        //********************************************
        // Device name: TS2-010CRM:WtrC-YCV-103
        // Device type: ICS_PV
        //********************************************

      "DEV_TS2-010CRM:WtrC-YCV-103_iDB" (EPICSToPLCLength:=5,
      EPICSToPLCDataBlockOffset:=55,
      PLCToEPICSLength:=34,
      PLCToEPICSDataBlockOffset:=137);

        //********************************************
        // Device name: TS2-010CRM:WtrC-YCV-104
        // Device type: ICS_PV
        //********************************************

      "DEV_TS2-010CRM:WtrC-YCV-104_iDB" (EPICSToPLCLength:=5,
      EPICSToPLCDataBlockOffset:=60,
      PLCToEPICSLength:=34,
      PLCToEPICSDataBlockOffset:=171);

        //********************************************
        // Device name: TS2-010CRM:WtrC-YSV-109
        // Device type: ICS_PV
        //********************************************

      "DEV_TS2-010CRM:WtrC-YSV-109_iDB" (EPICSToPLCLength:=5,
      EPICSToPLCDataBlockOffset:=65,
      PLCToEPICSLength:=34,
      PLCToEPICSDataBlockOffset:=205);

        //********************************************
        // Device name: TS2-010CRM:WtrC-YSV-110
        // Device type: ICS_PV
        //********************************************

      "DEV_TS2-010CRM:WtrC-YSV-110_iDB" (EPICSToPLCLength:=5,
      EPICSToPLCDataBlockOffset:=70,
      PLCToEPICSLength:=34,
      PLCToEPICSDataBlockOffset:=239);

        //********************************************
        // Device name: TS2-010CRM:WtrC-YSV-111
        // Device type: ICS_PV
        //********************************************

      "DEV_TS2-010CRM:WtrC-YSV-111_iDB" (EPICSToPLCLength:=5,
      EPICSToPLCDataBlockOffset:=75,
      PLCToEPICSLength:=34,
      PLCToEPICSDataBlockOffset:=273);

        //********************************************
        // Device name: TS2-010CRM:WtrC-YSV-112
        // Device type: ICS_PV
        //********************************************

      "DEV_TS2-010CRM:WtrC-YSV-112_iDB" (EPICSToPLCLength:=5,
      EPICSToPLCDataBlockOffset:=80,
      PLCToEPICSLength:=34,
      PLCToEPICSDataBlockOffset:=307);

        //********************************************
        // Device name: TS2-010CRM:WtrC-YSV-113
        // Device type: ICS_PV
        //********************************************

      "DEV_TS2-010CRM:WtrC-YSV-113_iDB" (EPICSToPLCLength:=5,
      EPICSToPLCDataBlockOffset:=85,
      PLCToEPICSLength:=34,
      PLCToEPICSDataBlockOffset:=341);

        //********************************************
        // Device name: TS2-010CRM:WtrC-TE-101
        // Device type: ICS_TT
        //********************************************

      "DEV_TS2-010CRM:WtrC-TE-101_iDB" (EPICSToPLCLength:=15,
      EPICSToPLCDataBlockOffset:=90,
      PLCToEPICSLength:=29,
      PLCToEPICSDataBlockOffset:=375);

        //********************************************
        // Device name: TS2-010CRM:WtrC-TE-102
        // Device type: ICS_TT
        //********************************************

      "DEV_TS2-010CRM:WtrC-TE-102_iDB" (EPICSToPLCLength:=15,
      EPICSToPLCDataBlockOffset:=105,
      PLCToEPICSLength:=29,
      PLCToEPICSDataBlockOffset:=404);

        //********************************************
        // Device name: TS2-010CRM:WtrC-TE-103
        // Device type: ICS_TT
        //********************************************

      "DEV_TS2-010CRM:WtrC-TE-103_iDB" (EPICSToPLCLength:=15,
      EPICSToPLCDataBlockOffset:=120,
      PLCToEPICSLength:=29,
      PLCToEPICSDataBlockOffset:=433);

        //********************************************
        // Device name: TS2-010CRM:WtrC-TE-104
        // Device type: ICS_TT
        //********************************************

      "DEV_TS2-010CRM:WtrC-TE-104_iDB" (EPICSToPLCLength:=15,
      EPICSToPLCDataBlockOffset:=135,
      PLCToEPICSLength:=29,
      PLCToEPICSDataBlockOffset:=462);
END_FUNCTION
DATA_BLOCK "EPICS_DebuggerResult"
{ S7_Optimized_Access := 'TRUE' }
VERSION : 0.1
NON_RETAIN
   VAR
      EPICS_Debugger_UtilitiesCall : String;   // PLCFactory Utilities call status
      EPICS_Debugger_DeviceCalls : String;   // PLCFactory DeviceCalls status
      EPICS_Debugger_IOCHash : String;   // EPICS IOC Hash vs. PLCFactory Hash
      EPICS_Debugger_ModBusHeartBeat : String;   // EPICS IOC Modbus (IOC->PLC) communication status
      EPICS_Debugger_S7Connection : String;   // EPICS IOC S7 TCP (PLC->IOC) communication status
      EPICS_Debugger_EPICS_GeneralState : String;   // Main status of the EPICS IOC communication
      EPICS_S7Port : Int;   // Actual TCP port that has been opened by the PLC
      EPICS_ModbusPort : Int;   // Actual ModBusTCP port that has been opened by the PLC
      EPICS_PLC_EthernetInterface : UInt;   // The currently used HW Identifer of the Ethernet Port on the PLC dedicated to EPICS
      EPICS_PayloadSize_InBytes : UInt;   // The currently configured payload size in bytes
      EPICS_PLC_Hash : DInt;   // The PLC Hash
      EPICS_PLCFactory_Version : String;   // The PLCFactory version that was used to generate the PLC code
      EPICS_CommunicationOK : Bool;   // Overall EPICS communication is OK
   END_VAR

BEGIN

END_DATA_BLOCK
FUNCTION_BLOCK "EPICS_DebuggerFB"
{ S7_Optimized_Access := 'TRUE' }
VERSION : 0.1
   VAR
      CheckUtilitiesTON {OriginalPartName := 'IEC_TIMER'; LibVersion := '1.0'; ExternalAccessible := 'False'; ExternalVisible := 'False'; ExternalWritable := 'False'} : TON_TIME;
      UtilSquareErrorTON { ExternalAccessible := 'False'; ExternalVisible := 'False'; ExternalWritable := 'False'} : Bool;
      CheckUtilitiesTON2 {OriginalPartName := 'IEC_TIMER'; LibVersion := '1.0'; ExternalAccessible := 'False'; ExternalVisible := 'False'; ExternalWritable := 'False'} : TON_TIME;
      UtilSquareErrorTON2 { ExternalAccessible := 'False'; ExternalVisible := 'False'; ExternalWritable := 'False'} : Bool;
      ModBus_TON {OriginalPartName := 'IEC_TIMER'; LibVersion := '1.0'; ExternalAccessible := 'False'; ExternalVisible := 'False'; ExternalWritable := 'False'} : TON_TIME;
      ModBus_wordsave { ExternalAccessible := 'False'; ExternalVisible := 'False'; ExternalWritable := 'False'} : Word;
   END_VAR
   VAR DB_SPECIFIC
      Helper_String { ExternalAccessible := 'False'; ExternalVisible := 'False'; ExternalWritable := 'False'} : String;
      Helper_String_Array { ExternalAccessible := 'False'; ExternalVisible := 'False'; ExternalWritable := 'False'} AT Helper_String : Struct
         String_Maximal { ExternalAccessible := 'False'; ExternalVisible := 'False'; ExternalWritable := 'False'} : Byte;
         String_Actual { ExternalAccessible := 'False'; ExternalVisible := 'False'; ExternalWritable := 'False'} : Byte;
         StringValueArray { ExternalAccessible := 'False'; ExternalVisible := 'False'; ExternalWritable := 'False'} : Array[0..15] of Byte;
      END_STRUCT;
   END_VAR
   VAR
      S7ConnTON {OriginalPartName := 'IEC_TIMER'; LibVersion := '1.0'; ExternalAccessible := 'False'; ExternalVisible := 'False'; ExternalWritable := 'False'} : TON_TIME;
   END_VAR

   VAR_TEMP
      AllOK { ExternalAccessible := 'False'; ExternalVisible := 'False'; ExternalWritable := 'False'} : Bool;
      i : Int;
      ModBusOK : Bool;
      S7OK : Bool;
   END_VAR


BEGIN
	//Author: Miklos Boros (miklos.boros@esss.se), Copyrigth 2017-2020 by European Spallation Source, Lund
	//This block was generated by PLCFactory
	//Description: This FB checks the EPICS configuration and outputs the result into EPICS_DebuggerResult.

	//DO NOT Modify this block!!!

	//AllOK will be evaluated in this code and passed to the EPICS_CommunicationOK signal that can be used by the PLC logic
	#AllOK := TRUE;

	#CheckUtilitiesTON(IN:="Utilities".Square_100ms,
	                   PT:=T#200ms,
	                   Q=>#UtilSquareErrorTON);

	#CheckUtilitiesTON2(IN := NOT "Utilities".Square_100ms,
	                   PT := T#200ms,
	                   Q => #UtilSquareErrorTON2);


	#ModBus_TON(IN := #ModBus_wordsave = "EPICSToPLC"."Word"[2],
	            PT := T#5s);


     "EPICS_DebuggerResult".#EPICS_PayloadSize_InBytes := 982;
     "EPICS_DebuggerResult".#EPICS_PLC_Hash := -1975058360;
     "EPICS_DebuggerResult".#EPICS_PLCFactory_Version := 'ffa943c824bc42c5378196579606b0f20e8dd5c8';

	IF ("Utilities".AlwaysOn = FALSE) THEN
	    "EPICS_DebuggerResult".#EPICS_Debugger_UtilitiesCall := 'ERROR: FunctionBlock: "_UilitiesFB" is called with a wrong InstanceDB. Call it with the existing iDB named: "Utilities" AND check if the System Memory bits and the System Clock byte is enabled!';
         #AllOK := FALSE;
	ELSE
	    IF (#UtilSquareErrorTON OR #UtilSquareErrorTON2) THEN
	        "EPICS_DebuggerResult".#EPICS_Debugger_UtilitiesCall := 'ERROR: FunctionBlock: "_UilitiesFB" is called with a wrong InstanceDB. Call it with the existing iDB named: "Utilities" AND check if the System Memory bits and the System Clock byte is enabled!';
             #AllOK := FALSE;
	    ELSE
	        "EPICS_DebuggerResult".#EPICS_Debugger_UtilitiesCall := 'OK: EPICS Utilities works as expected.';

	    END_IF;
	END_IF;

	IF ("Utilities".EPICS_Device_calls_precessed) THEN
	    "EPICS_DebuggerResult".#EPICS_Debugger_DeviceCalls := 'OK: "EPICS_device_calls" is called as expected.';
	ELSE
	    "EPICS_DebuggerResult".#EPICS_Debugger_DeviceCalls := 'ERROR: "EPICS_device_calls" is not called in OB1!';
         #AllOK := FALSE;
	END_IF;

	IF (("EPICSToPLC"."Word"[0] = "PLCToEPICS"."Word"[0]) AND ("EPICSToPLC"."Word"[1] = "PLCToEPICS"."Word"[1])) THEN
	    "EPICS_DebuggerResult".#EPICS_Debugger_IOCHash := 'OK: IOC and PLC hash are equal.';
	ELSE
	    "EPICS_DebuggerResult".#EPICS_Debugger_IOCHash := 'ERROR: IOC and PLC hash are NOT equal!';
         #AllOK := FALSE;
	END_IF;

	IF (#ModBus_TON.Q) THEN
	    "EPICS_DebuggerResult".#EPICS_Debugger_ModBusHeartBeat := 'ERROR: The IOC is not sending any HeartBeat via ModBus!';
         #AllOK := FALSE;
	    #ModBusOK := FALSE;
	ELSE
	    "EPICS_DebuggerResult".#EPICS_Debugger_ModBusHeartBeat := 'OK: ModBus HeartBeat is received as expected.';
	    #ModBusOK := TRUE;
	END_IF;

	#S7ConnTON(IN := NOT "_CommsPLC_EPICS_DB".SendDone, PT := T#3s);

	IF ("_CommsPLC_EPICS_DB".BytesToSend > 0) THEN

	    IF (#S7ConnTON.Q) THEN
	        "EPICS_DebuggerResult".EPICS_Debugger_S7Connection := 'ERROR: EPICS S7 connection can not send Status variables!';
	        #S7OK := FALSE;
             #AllOK := FALSE;
	    ELSE
	        "EPICS_DebuggerResult".EPICS_Debugger_S7Connection := 'OK: EPICS S7 works as expected.';
	        #S7OK := TRUE;

	    END_IF;
	ELSE
	    "EPICS_DebuggerResult".EPICS_Debugger_S7Connection := 'OK: EPICS S7 disabled, there is no Status variable to send.';
	    #S7OK := TRUE;
	END_IF;

	IF (#ModBusOK AND #S7OK) THEN
	    "EPICS_DebuggerResult".EPICS_Debugger_EPICS_GeneralState := 'OK. EPICS IOC communication is ONLINE.';
	END_IF;

	IF (#ModBusOK AND NOT #S7OK) THEN
	    "EPICS_DebuggerResult".EPICS_Debugger_EPICS_GeneralState := 'ERROR. ModBus seems to be working but S7 TCP is blocked. Try to check your PLC router IP.';
         #AllOK := FALSE;
	END_IF;

	IF (NOT #ModBusOK AND #S7OK) THEN
	    "EPICS_DebuggerResult".EPICS_Debugger_EPICS_GeneralState := 'ERROR. ModBus seems to be offline. Waiting for IOC to finish connecting to the PLC.';
         #AllOK := FALSE;
	END_IF;

	IF ( NOT #ModBusOK AND NOT #S7OK) THEN
	    "EPICS_DebuggerResult".EPICS_Debugger_EPICS_GeneralState := 'ERROR. Both ModBus and S7 TCP seems to be offline. Check if your IOC is running and if it is connected to the right PLC interface. Your HardwareID comes from CCDB!';
         #AllOK := FALSE;
	END_IF;

	"EPICS_DebuggerResult".EPICS_ModbusPort := "_CommsPLC_EPICS_DB".MBPort;
	"EPICS_DebuggerResult".EPICS_S7Port := "_CommsPLC_EPICS_DB".S7Port;
	"EPICS_DebuggerResult".EPICS_PLC_EthernetInterface :=  "_CommsPLC_EPICS_DB".InterfaceID;

	#ModBus_wordsave := "EPICSToPLC"."Word"[2];

	//Put the Overall result to the Globl DB
	"EPICS_DebuggerResult".EPICS_CommunicationOK := #AllOK;


END_FUNCTION_BLOCK
DATA_BLOCK "EPICS_DebuggerFB_iDB"
{ S7_Optimized_Access := 'TRUE' }
VERSION : 0.1
NON_RETAIN
"EPICS_DebuggerFB"

BEGIN

END_DATA_BLOCK
ORGANIZATION_BLOCK "EPICS_DebuggerOB"
TITLE = "Main Program Sweep (Cycle)"
{ S7_Optimized_Access := 'TRUE' }
VERSION : 0.1

BEGIN
	//Author: Miklos Boros (miklos.boros@esss.se), Copyrigth 2017-2020 by European Spallation Source, Lund
	//This block was generated by PLCFactory
	//Description: This OB is a cyclic OB called in every PLC cycle and EPICS_DebuggerFB checks the EPICS configuration.

	//DO NOT Modify this block!!!
	"EPICS_DebuggerFB_iDB"();


END_ORGANIZATION_BLOCK
DATA_BLOCK "EPICSToPLC"
{ S7_Optimized_Access := 'FALSE' }
VERSION : 0.1
//########## EPICS->PLC datablock ##########
   STRUCT
      "Word" { ExternalAccessible := 'False'; ExternalVisible := 'False'; ExternalWritable := 'False'; } : Array[0..149] of Word;
   END_STRUCT;

BEGIN

END_DATA_BLOCK

DATA_BLOCK "PLCToEPICS"
{ S7_Optimized_Access := 'FALSE' }
VERSION : 0.1
NON_RETAIN
//########## PLC->EPICS datablock ##########
   STRUCT
      "Word" { ExternalAccessible := 'False'; ExternalVisible := 'False'; ExternalWritable := 'False'; } : Array[0..490] of Word;
   END_STRUCT;

BEGIN

END_DATA_BLOCK

FUNCTION "_CommsEPICS" : Void
{ S7_Optimized_Access := 'TRUE' }
VERSION : 0.1
   VAR_TEMP
      PLC_Hash : DInt;
   END_VAR

BEGIN
	//Heartbeat PLC->EPICS
	IF "Utilities".Pulse_1s THEN
	    "PLCToEPICS"."Word"[2] := "PLCToEPICS"."Word"[2] + 1;
	    IF "PLCToEPICS"."Word"[2] >= 32000 THEN
	        "PLCToEPICS"."Word"[2] := 0;
	    END_IF;
	END_IF;

	// PLC Factory commit ID: ffa943c824bc42c5378196579606b0f20e8dd5c8
	// PLC Hash (Generated by PLC Factory)
	#PLC_Hash := DINT#-1975058360;

	// Send the PLC Hash to the EPICS IOC
	"PLCToEPICS"."Word"[1] := DINT_TO_WORD(#PLC_Hash);
	"PLCToEPICS"."Word"[0] := DINT_TO_WORD(SHR(IN := #PLC_Hash, N := 16));

	// Send the PLC parameter upload status to the EPICS IOC
	"PLCToEPICS"."Word"[3] := "EPICSToPLC"."Word"[5];
     "Utilities".EPICSParametersStatus := "EPICSToPLC"."Word"[5];

	// Put the PLC Hash into the Modbus map
	"EPICSToPLC"."Word"[4] := DINT_TO_WORD(#PLC_Hash);
	"EPICSToPLC"."Word"[3] := DINT_TO_WORD(SHR(IN := #PLC_Hash, N := 16));


	// Put the payload size (in bytes) into the Modbus map
	"EPICSToPLC"."Word"[6] := 982;

	// Call the comms block to provide PLC<->EPICS comms
	"_CommsPLC_EPICS_DB"(Enable         := "Utilities".AlwaysOn,
	                     SendTrigger    := "Utilities".Pulse_200ms,
	                     BytesToSend    := 982,
	                     InterfaceID    := 72,
	                     S7ConnectionID := 256,
	                     MBConnectionID := 255,
	                     S7Port         := 2000,
	                     MBPort         := 502,
	                     PLCToEPICSData := "PLCToEPICS"."Word",
	                     EPICSToPLCData := "EPICSToPLC"."Word");

END_FUNCTION
